# EPICS substitutions: db/Beckhoff_3XXX/ecmcEL3602.substitutions
file "ecmc_analogInput-chX.template"
{
  pattern {CH_ID, ESLO, EOFF, EGU, PREC}
          {01, "${_ESLO=4.656612875E-9}", "${_EOFF=0}", "${_EGU=V}", "${_PREC=3}"}
          {02, "${_ESLO=4.656612875E-9}", "${_EOFF=0}", "${_EGU=V}", "${_PREC=3}"}
}

file "ecmc_status_analog-chX.template"
{
  pattern {CH_ID, KEY }
          {01,    "AI"}
          {02,    "AI"}
}
